FUNCTION_BLOCK SecuringWorkpiece
VAR_INPUT
	MethodCall : BOOL;
	TS_Endschalter_01: BOOL;
	TS_Endschalter_02: BOOL;
	SecuringTime : TIME;
	NotAusSignal : BOOL;
	AutomaticMode: BOOL;
END_VAR
VAR_OUTPUT
	SecuringProcess : BOOL;
END_VAR
VAR
//FlipFlop
	RS_SecuringProcessON: RS;	
//Zeitverzögerung
	TON_SecuringTime: TON;
//Flanke	
	R_TRIG_MethodCall: R_TRIG;
END_VAR

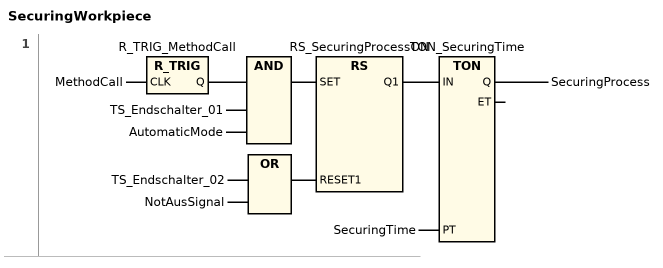
// NETWORK 1
R_TRIG_MethodCall(CLK := MethodCall); // R_TRIG
RS_SecuringProcessON(SET := R_TRIG_MethodCall.Q AND TS_Endschalter_01 AND AutomaticMode, RESET1 := TS_Endschalter_02 OR NotAusSignal); // RS
TON_SecuringTime(IN := RS_SecuringProcessON.Q1, PT := SecuringTime); // TON
SecuringProcess := TON_SecuringTime.Q;

END_FUNCTION_BLOCK

(* stored: Version 1.1.0.1, ProductVersion 3.1.4024.15
   POU SecuringWorkpiece: Id {9cafd3de-dbf0-474b-af08-30a8d1cbba1a}, SpecialFunc None *)
